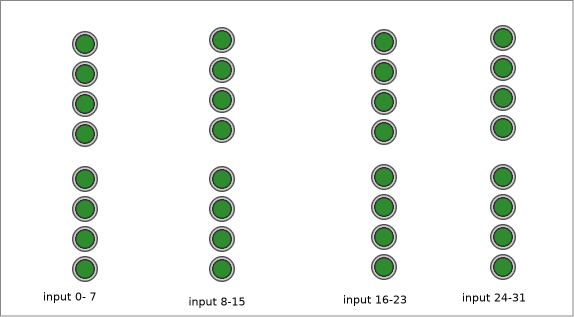
VISUALIZATION InitSoftware  // 574x317
    Lamp1 (69,29 32x30), variable: GVL.I_Input00, style: Lamp-Lamp1-Green
    Lamp1 (69,59 32x30), variable: GVL.I_Input01, style: Lamp-Lamp1-Green
    Lamp1 (69,89 32x30), variable: GVL.I_Input02, style: Lamp-Lamp1-Green
    Lamp1 (69,119 32x30), variable: GVL.I_Input03, style: Lamp-Lamp1-Green
    Lamp1 (69,164 32x30), variable: GVL.I_Input04, style: Lamp-Lamp1-Green
    Lamp1 (69,194 32x30), variable: GVL.I_Input05, style: Lamp-Lamp1-Green
    Lamp1 (69,224 32x30), variable: GVL.I_Input06, style: Lamp-Lamp1-Green
    Lamp1 (69,254 32x30), variable: GVL.I_Input07, style: Lamp-Lamp1-Green
    Lamp1 (206,25 32x30), variable: GVL.I_Input08, style: Lamp-Lamp1-Green
    Lamp1 (206,55 32x30), variable: GVL.I_Input09, style: Lamp-Lamp1-Green
    Lamp1 (206,85 32x30), variable: GVL.I_Input10, style: Lamp-Lamp1-Green
    Lamp1 (206,115 32x30), variable: GVL.I_Input11, style: Lamp-Lamp1-Green
    Lamp1 (206,164 32x30), variable: GVL.I_Input12, style: Lamp-Lamp1-Green
    Lamp1 (206,194 32x30), variable: GVL.I_Input13, style: Lamp-Lamp1-Green
    Lamp1 (206,224 32x30), variable: GVL.I_Input14, style: Lamp-Lamp1-Green
    Lamp1 (206,254 32x30), variable: GVL.I_Input15, style: Lamp-Lamp1-Green
    Lamp1 (368,27 32x30), variable: GVL.I_Input16, style: Lamp-Lamp1-Green
    Lamp1 (368,57 32x30), variable: GVL.I_Input17, style: Lamp-Lamp1-Green
    Lamp1 (368,87 32x30), variable: GVL.I_Input18, style: Lamp-Lamp1-Green
    Lamp1 (368,117 32x30), variable: GVL.I_Input19, style: Lamp-Lamp1-Green
    Lamp1 (368,162 32x30), variable: GVL.I_Input20, style: Lamp-Lamp1-Green
    Lamp1 (368,192 32x30), variable: GVL.I_Input21, style: Lamp-Lamp1-Green
    Lamp1 (368,222 32x30), variable: GVL.I_Input22, style: Lamp-Lamp1-Green
    Lamp1 (368,252 32x30), variable: GVL.I_Input23, style: Lamp-Lamp1-Green
    Lamp1 (487,23 32x30), variable: GVL.I_Input24, style: Lamp-Lamp1-Green
    Lamp1 (487,53 32x30), variable: GVL.I_Input25, style: Lamp-Lamp1-Green
    Lamp1 (487,83 32x30), variable: GVL.I_Input26, style: Lamp-Lamp1-Green
    Lamp1 (487,113 32x30), variable: GVL.I_Input27, style: Lamp-Lamp1-Green
    Lamp1 (487,162 32x30), variable: GVL.I_Input28, style: Lamp-Lamp1-Green
    Lamp1 (487,192 32x30), variable: GVL.I_Input29, style: Lamp-Lamp1-Green
    Lamp1 (487,222 32x30), variable: GVL.I_Input30, style: Lamp-Lamp1-Green
    Lamp1 (487,252 32x30), variable: GVL.I_Input31, style: Lamp-Lamp1-Green
    Label (-5,282 150x30), "input 0- 7"
    Label (300,285 150x30), "input 16-23"
    Label (142,287 150x30), "input 8-15"
    Label (419,283 150x30), "input 24-31"
END_VISUALIZATION

(* stored: Version 1.1.0.1, ProductVersion 3.1.4024.11
   Visu InitSoftware: Id {5e66dc43-631d-4728-9682-911be535eba1} *)
